// TIA Portal V17 export
// export: Created 2025-03-05T08:00:22.1000979Z, ExportSetting WithDefaults, DisplayName Totally Integrated Automation Portal, DisplayVersion V17 Update 8, DisplayName TIA Portal Openness, DisplayVersion V17 Update 8, DisplayName TIA Portal Version Control Interface, DisplayVersion V17, DisplayName SINAMICS Startdrive Advanced, DisplayVersion V17 SP2, DisplayName SINAMICS Startdrive G110M, G120, G120C, G120D, G120P, G115D, DisplayVersion V17 SP2, DisplayName SINAMICS Startdrive G130, G150, S120, S150, SINAMICS MV, S210, DisplayVersion V17 SP2, DisplayName STEP 7 Professional, DisplayVersion V17 Update 8, DisplayName SINUMERIK ONE STEP 7 Toolbox, DisplayVersion V17 Update 12, DisplayName SINUMERIK 840D sl STEP 7 Toolbox, DisplayVersion V17 Update 12, DisplayName STEP 7 Safety, DisplayVersion V17 Update 6, DisplayName WinCC Advanced, DisplayVersion V17 Update 8
DATA_BLOCK "DB130_SPINDLE_AXIS_OPTIONS"   // DB130
{ S7_Optimized_Access := 'TRUE'; DB_Accessible_From_OPC_UA := 'FALSE' }
VERSION : 0.1
// stored: AutoNumber false, DBAccessibleFromOPCUA false, DBAccessibleFromWebserver true, IsOnlyStoredInLoadMemory false, IsRetainMemResEnabled false, IsWriteProtectedInAS false, MemoryReserve 100
   VAR
      C11_AXIS_SPINDLE_MODE : Bool;   // C11 AXIS SPINDLE (V) MODE CONFIGURED
      C12_AXIS_SPINDLE_MODE : Bool;   // C12 AXIS SPINDLE (V) MODE CONFIGURED
      C13_AXIS_SPINDLE_MODE : Bool;   // C13 AXIS SPINDLE (V) MODE CONFIGURED
      C14_AXIS_SPINDLE_MODE : Bool;   // C14 AXIS SPINDLE (V) MODE CONFIGURED
      C21_AXIS_SPINDLE_MODE : Bool;   // C21 AXIS SPINDLE (V) MODE CONFIGURED
      C22_AXIS_SPINDLE_MODE : Bool;   // C22 AXIS SPINDLE (V) MODE CONFIGURED
      C23_AXIS_SPINDLE_MODE : Bool;   // C23 AXIS SPINDLE (V) MODE CONFIGURED
      C24_AXIS_SPINDLE_MODE : Bool;   // C24 AXIS SPINDLE (V) MODE CONFIGURED
      C31_AXIS_SPINDLE_MODE : Bool;   // C24 AXIS SPINDLE (V) MODE CONFIGURED
   END_VAR
BEGIN
END_DATA_BLOCK
